INTERFACE I_InputPortAddedEvent EXTENDS I_Event

PROPERTY PUBLIC Target : I_InputPort
GET
END_GET
END_PROPERTY

END_INTERFACE

(* stored: Version 1.1.0.1, ProductVersion 3.1.4024.12
   Itf I_InputPortAddedEvent: Id {4240fb31-aed0-0eb8-1c7b-44efaab6ad65}
   Property Target: Id {21689131-12f2-0420-2b3e-b602a0e9f23b}
   Get Get: Id {969e48c5-2057-0376-054d-cd274e160896} *)
